// TIA Portal V20 export
TYPE "IO_Device_Test_Parameters_Rework"
   STRUCT
      Reset_PLC_Functional_Test_Rework : Bool;
      Status : Bool;
      Voltage_Read : UInt;
      Min_Electrical_Current : UInt;
      Max_Electrical_Current : UInt;
      Time_End_Electrical_Current_Test : Time;
      Time_Start_Visual_Test : Time;
   END_STRUCT;
END_TYPE
